// LS Electric XG5000 project: 8_26_데이터 전송 명령
// PLC LSPLC
// module base 0 slot 0: 입출력 모듈:XBC-DN/DP14E (DC 24V 입력 8점, 트랜지스터 출력 6점)

PROGRAM NewProgram (task: 스캔 프로그램)

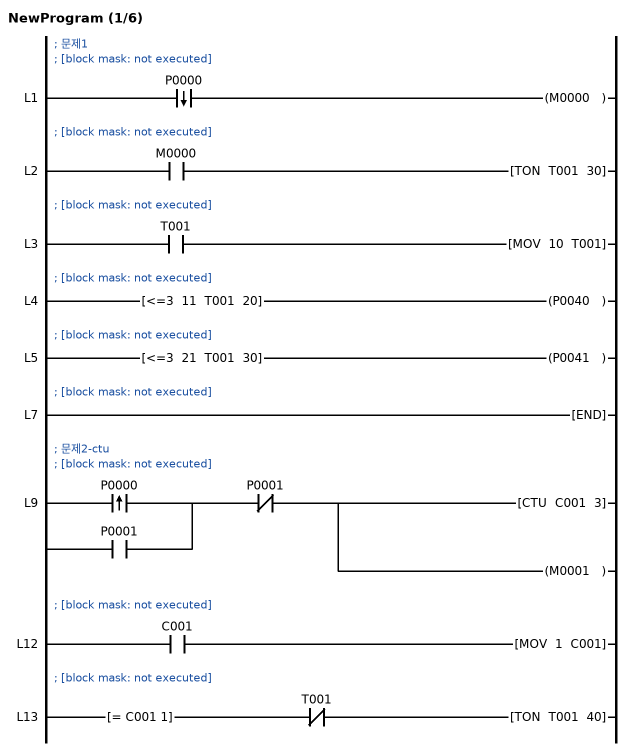
// 문제1
; L1 (block mask: not executed)
LOADN     P0000
OUT       M0000
; L2 (block mask: not executed)
LOAD      M0000
TON       T001 30
; L3 (block mask: not executed)
LOAD      T001
MOV       10 T001
; L4 (block mask: not executed)
LOAD<=3   11 T001 20
OUT       P0040
; L5 (block mask: not executed)
LOAD<=3   21 T001 30
OUT       P0041
; L7 (block mask: not executed)
END
// 문제2-ctu
; L9 (block mask: not executed)
LOADP     P0000
OR        P0001
AND NOT   P0001
CTU       C001 3
OUT       M0001
; L12 (block mask: not executed)
LOAD      C001
MOV       1 C001
; L13 (block mask: not executed)
LOAD=     C001 1
AND NOT   T001
TON       T001 40

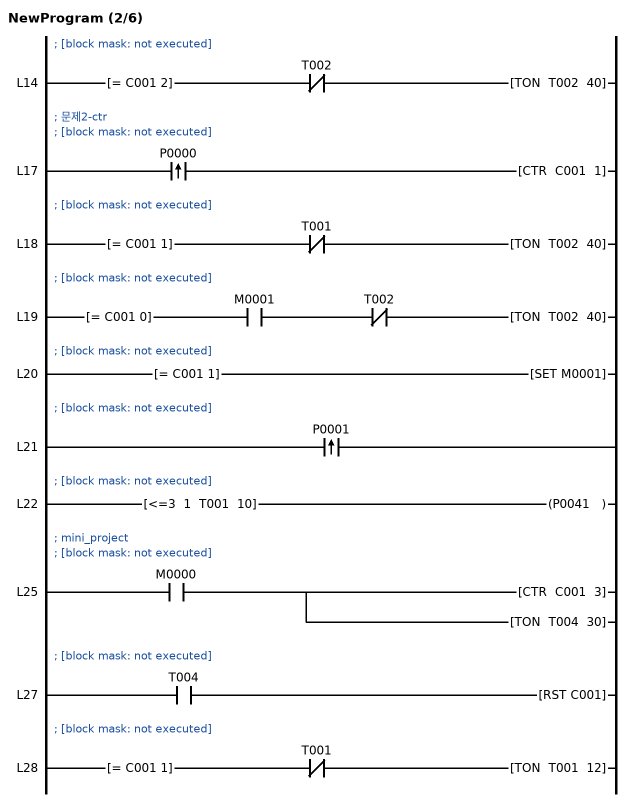
; L14 (block mask: not executed)
LOAD=     C001 2
AND NOT   T002
TON       T002 40
// 문제2-ctr
; L17 (block mask: not executed)
LOADP     P0000
CTR       C001 1
; L18 (block mask: not executed)
LOAD=     C001 1
AND NOT   T001
TON       T002 40
; L19 (block mask: not executed)
LOAD=     C001 0
AND       M0001
AND NOT   T002
TON       T002 40
; L20 (block mask: not executed)
LOAD=     C001 1
SET       M0001
; L21 (block mask: not executed)
LOADP     P0001
; L22 (block mask: not executed)
LOAD<=3   1 T001 10
OUT       P0041
// mini_project
; L25 (block mask: not executed)
LOAD      M0000
CTR       C001 3
TON       T004 30
; L27 (block mask: not executed)
LOAD      T004
RST       C001
; L28 (block mask: not executed)
LOAD=     C001 1
AND NOT   T001
TON       T001 12

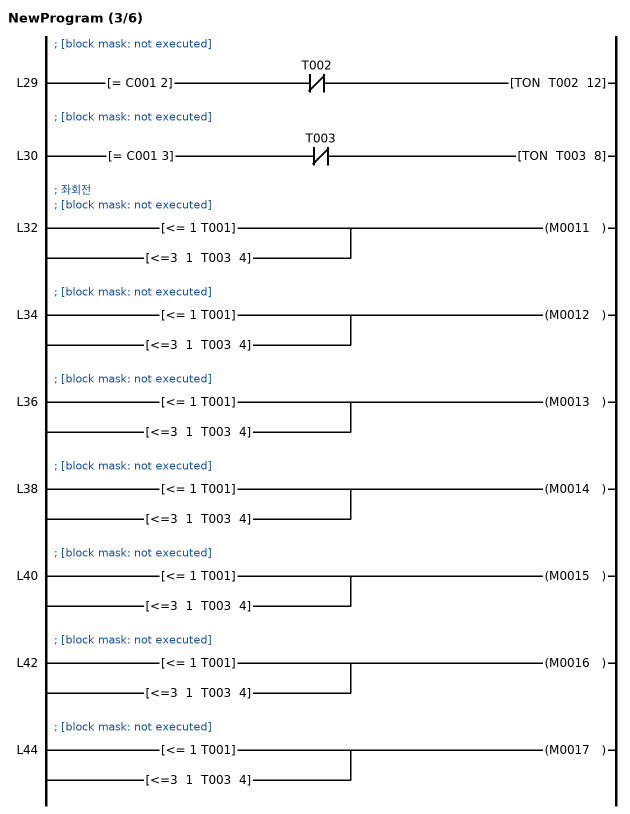
; L29 (block mask: not executed)
LOAD=     C001 2
AND NOT   T002
TON       T002 12
; L30 (block mask: not executed)
LOAD=     C001 3
AND NOT   T003
TON       T003 8
// 좌회전
; L32 (block mask: not executed)
LOAD<=    1 T001
OR<=3     1 T003 4
OUT       M0011
; L34 (block mask: not executed)
LOAD<=    1 T001
OR<=3     1 T003 4
OUT       M0012
; L36 (block mask: not executed)
LOAD<=    1 T001
OR<=3     1 T003 4
OUT       M0013
; L38 (block mask: not executed)
LOAD<=    1 T001
OR<=3     1 T003 4
OUT       M0014
; L40 (block mask: not executed)
LOAD<=    1 T001
OR<=3     1 T003 4
OUT       M0015
; L42 (block mask: not executed)
LOAD<=    1 T001
OR<=3     1 T003 4
OUT       M0016
; L44 (block mask: not executed)
LOAD<=    1 T001
OR<=3     1 T003 4
OUT       M0017

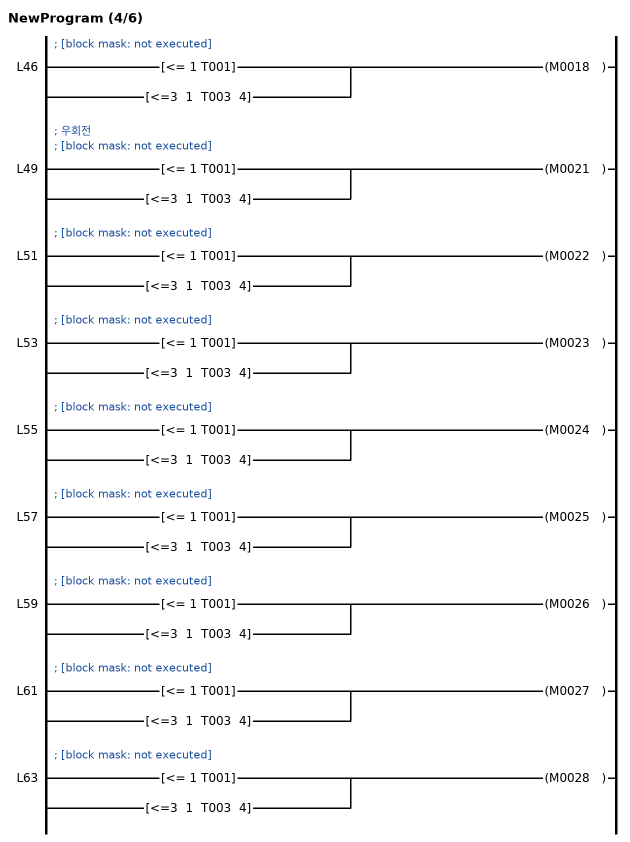
; L46 (block mask: not executed)
LOAD<=    1 T001
OR<=3     1 T003 4
OUT       M0018
// 우회전
; L49 (block mask: not executed)
LOAD<=    1 T001
OR<=3     1 T003 4
OUT       M0021
; L51 (block mask: not executed)
LOAD<=    1 T001
OR<=3     1 T003 4
OUT       M0022
; L53 (block mask: not executed)
LOAD<=    1 T001
OR<=3     1 T003 4
OUT       M0023
; L55 (block mask: not executed)
LOAD<=    1 T001
OR<=3     1 T003 4
OUT       M0024
; L57 (block mask: not executed)
LOAD<=    1 T001
OR<=3     1 T003 4
OUT       M0025
; L59 (block mask: not executed)
LOAD<=    1 T001
OR<=3     1 T003 4
OUT       M0026
; L61 (block mask: not executed)
LOAD<=    1 T001
OR<=3     1 T003 4
OUT       M0027
; L63 (block mask: not executed)
LOAD<=    1 T001
OR<=3     1 T003 4
OUT       M0028

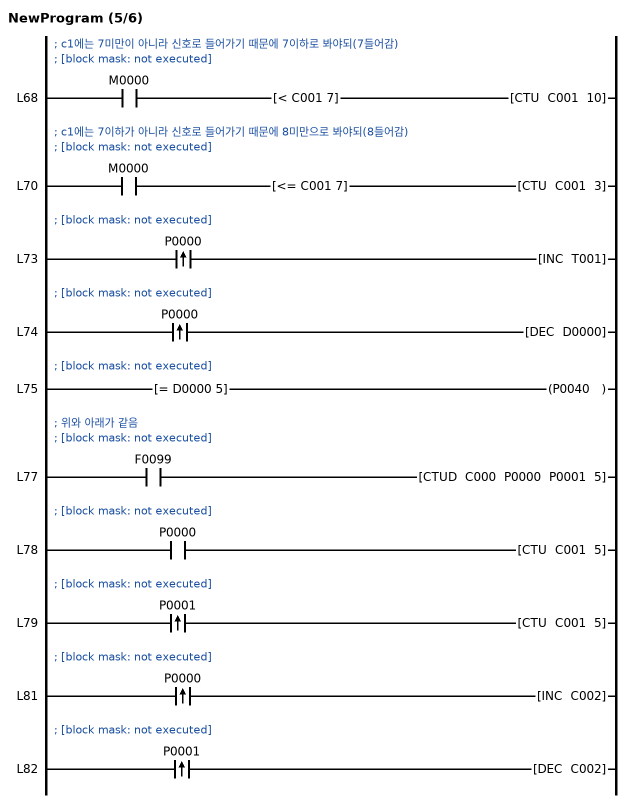
// c1에는 7미만이 아니라 신호로 들어가기 때문에 7이하로 봐야되(7들어감)
; L68 (block mask: not executed)
LOAD      M0000
AND<      C001 7
CTU       C001 10
// c1에는 7이하가 아니라 신호로 들어가기 때문에 8미만으로 봐야되(8들어감)
; L70 (block mask: not executed)
LOAD      M0000
AND<=     C001 7
CTU       C001 3
; L73 (block mask: not executed)
LOADP     P0000
INC       T001
; L74 (block mask: not executed)
LOADP     P0000
DEC       D0000
; L75 (block mask: not executed)
LOAD=     D0000 5
OUT       P0040
// 위와 아래가 같음
; L77 (block mask: not executed)
LOAD      F0099
CTUD      C000 P0000 P0001 5
; L78 (block mask: not executed)
LOAD      P0000
CTU       C001 5
; L79 (block mask: not executed)
LOADP     P0001
CTU       C001 5
; L81 (block mask: not executed)
LOADP     P0000
INC       C002
; L82 (block mask: not executed)
LOADP     P0001
DEC       C002

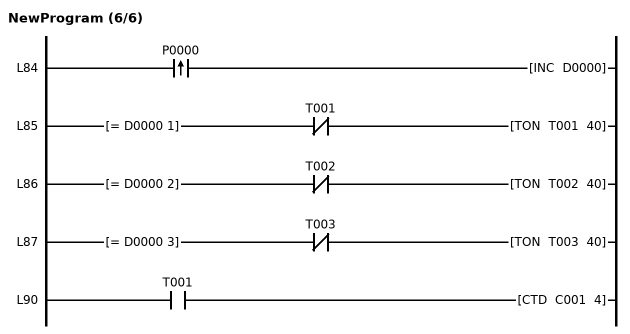
; L84
LOADP     P0000
INC       D0000
; L85
LOAD=     D0000 1
AND NOT   T001
TON       T001 40
; L86
LOAD=     D0000 2
AND NOT   T002
TON       T002 40
; L87
LOAD=     D0000 3
AND NOT   T003
TON       T003 40
; L90
LOAD      T001
CTD       C001 4